# B&R Automation Studio project 3964r
Automation Studio 4.2.8.54 SP

## Configuration cp1381

CPU X20CP1381, AutomationRuntime B4.26, Build 4.1.2, Vc V4.26.2

CPU X20CP3586, AutomationRuntime B4.26, Build 4.1.2, Vc V4.26.2

### Task classes (Cpu.sw)
```
Cyclic#1 (cycle 10000 us, tolerance 10000 us):
  3964r1 <- 3964r.prg
Binaries: TCData, arconfig, asfw, ashwd, iomap, asnxdb1, User, Role, sysconf
Libraries: DRV_3964, dvframe, runtime, asstring, standard, astime, asieccon, IecCheck, sys_lib, AsBrStr
```

### Hardware
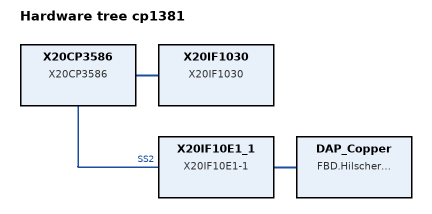
```
DAP_Copper : FBD.Hilscher.PNIOGenDevDTM2.DAP Copper.V1.09.05 v1.9.5 (OrderNumber=DAP Copper)  [PN1 -> X20IF10E1_1.IF1 (NodeNumber=1)]
  DtmId = 207df88f-8d0b-476b-a90a-ff4e51565477
  DtmRef = FBD.Hilscher.PNIOGenDevDTM2.DAP Copper.V1.09.05
  ChannelBlocks_54764a2b-737d-4760-b2ae-f15fab32f69c  // Retrofit Image <Slot 1>
  IO_InputImage_54764a2b-737d-4760-b2ae-f15fab32f69c
  IO_OutputImage_54764a2b-737d-4760-b2ae-f15fab32f69c
X20CP3586 : X20CP3586 v1.3.2.0
  Connector IF2:
    ActivateDevice = 1
    EthInterfaceRedundant = 0
    Mode = Manual
    InternetAddress = 192.168.20.10
    SubnetMask = 255.255.255.0
  Connector IF3:
    EplInterfaceRedundant = 0
    CycleTime = 10000
    EplEthInterfaceRedundant = 0
  ConfigurationID = test1_cp1381
  TimerDeviceType = SWIOTIMER
  Cyclic1Duration = 10000
  Cyclic1Tolerance = 10000
  Cyclic2Duration = 20000
  Cyclic2Tolerance = 20000
  Cyclic3Duration = 10000
  Cyclic3Tolerance = 50000
  Cyclic4Duration = 100000
  Cyclic4Tolerance = 100000
  Cyclic5Duration = 200000
  Cyclic5Tolerance = 200000
  Cyclic6Duration = 500000
  Cyclic6Tolerance = 500000
  Cyclic7Duration = 1000000
  Cyclic7Tolerance = 1000000
  Cyclic8Duration = 10000
  Cyclic8Tolerance = 30000000
X20IF1030 : X20IF1030 v1.1.7.0  [SS -> X20CP3586.SS1]
X20IF10E1_1 : X20IF10E1-1 v1.1.5.0  [SS -> X20CP3586.SS2]
  Connector IF1:
    DtmRef = FBDIF.Hilscher.PNIOControllerDTM2.NETX 100 RE/PNM
    DtmId = 1afa87f6-e739-4a4c-a598-27084086dda1
  ConfigFile = X20IF10E1_1.dtm
  ConfigModule = asnxdb1
```

### IoMap.iom - X20CP3586/IoMap.iom
```iecst
VAR_CONFIG
	::3964r1:profinetInput1[0] AT %IB."DAP_Copper".Module001_Input8_00;
	::3964r1:profinetInput1[1] AT %IB."DAP_Copper".Module001_Input8_01;
	::3964r1:profinetInput1[2] AT %IB."DAP_Copper".Module001_Input8_02;
	::3964r1:profinetInput1[3] AT %IB."DAP_Copper".Module001_Input8_03;
	::3964r1:profinetOutput1[0] AT %QB."DAP_Copper".Module001_Output8_00;
	::3964r1:profinetOutput1[1] AT %QB."DAP_Copper".Module001_Output8_01;
	::3964r1:profinetOutput1[2] AT %QB."DAP_Copper".Module001_Output8_02;
	::3964r1:profinetOutput1[3] AT %QB."DAP_Copper".Module001_Output8_03;
	::3964r1:profinetInput2[0] AT %IB."DAP_Copper".Module001_Input_00;
	::3964r1:profinetInput2[1] AT %IB."DAP_Copper".Module001_Input_01;
	::3964r1:profinetInput2[2] AT %IB."DAP_Copper".Module001_Input_02;
	::3964r1:profinetInput2[3] AT %IB."DAP_Copper".Module001_Input_03;
	::3964r1:profinetInput2[4] AT %IB."DAP_Copper".Module001_Input_04;
	::3964r1:profinetInput2[5] AT %IB."DAP_Copper".Module001_Input_05;
	::3964r1:profinetInput2[6] AT %IB."DAP_Copper".Module001_Input_06;
	::3964r1:profinetInput2[7] AT %IB."DAP_Copper".Module001_Input_07;
	::3964r1:profinetInput2[8] AT %IB."DAP_Copper".Module001_Input_08;
	::3964r1:profinetInput2[9] AT %IB."DAP_Copper".Module001_Input_09;
	::3964r1:profinetInput2[10] AT %IB."DAP_Copper".Module001_Input_10;
	::3964r1:profinetOutput2[0] AT %QB."DAP_Copper".Module001_Output_00;
	::3964r1:profinetOutput2[1] AT %QB."DAP_Copper".Module001_Output_01;
	::3964r1:profinetOutput2[2] AT %QB."DAP_Copper".Module001_Output_02;
	::3964r1:profinetOutput2[3] AT %QB."DAP_Copper".Module001_Output_03;
	::3964r1:profinetOutput2[4] AT %QB."DAP_Copper".Module001_Output_04;
	::3964r1:profinetOutput2[5] AT %QB."DAP_Copper".Module001_Output_05;
	::3964r1:profinetOutput2[6] AT %QB."DAP_Copper".Module001_Output_06;
	::3964r1:profinetOutput2[7] AT %QB."DAP_Copper".Module001_Output_07;
	::3964r1:profinetOutput2[8] AT %QB."DAP_Copper".Module001_Output_08;
	::3964r1:profinetOutput2[9] AT %QB."DAP_Copper".Module001_Output_09;
	::3964r1:profinetOutput2[10] AT %QB."DAP_Copper".Module001_Output_10;
END_VAR
```

## Logical view

Binary libraries used (declarations not repeated): operator, runtime, astime, AsIecCon, DRV_3964, dvframe, asstring, standard, sys_lib, AsBrStr

### Package Logical/Libraries - Global libraries

### Library Logical/Libraries/IecCheck (IEC)
Depends on: sys_lib, AsBrStr

### Program Logical/3964r (IEC)

#### Types.typ
```iecst
TYPE
	FromFronius : 	STRUCT
		arcStable : BOOL;
		processActive : BOOL;
		mainCurrentSignal : BOOL;
		torchCollisionProtection : BOOL;
		powerSourceReady : BOOL;
		communicationReady : BOOL;
		powerOutsideRange : BOOL;
		weldingVoltageActual : UINT;
		weldingCurrentActual : UINT;
		wireFeedSpeed : UINT;
	END_STRUCT;
	FromComau : 	STRUCT
		weldingStart : BOOL;
		robotReady : BOOL;
		modesBit0 : BOOL;
		modesBit1 : BOOL;
		modesBit2 : BOOL;
		gasTest : BOOL;
		wireInching : BOOL;
		wireRetract : BOOL;
		touchSensing : BOOL;
		torchBlowOut : BOOL;
		jobNumber : USINT;
		weldingSimulation : BOOL;
		powerCommand : UINT;
		arcLengthCorrection : UINT;
		pulseCorrection : USINT;
		burnBackCommand : USINT;
		synchroPulseDisable : BOOL;
		temp : ARRAY[0..19]OF USINT;
	END_STRUCT;
	Interface3964R : 	STRUCT
		fromComau : FromComau;
		fromFronius : FromFronius;
	END_STRUCT;
END_TYPE
```

#### Variables.var
```iecst
VAR
	interface3964R : Interface3964R;
	step : INT;
	FRM_xopen_0 : FRM_xopen;
	FRM_read_0 : FRM_read;
	dataRead : ARRAY[0..19] OF USINT;
	FRM_rbuf_0 : FRM_rbuf;
	dataReadLength : INT;
	FRM_gbuf_0 : FRM_gbuf;
	FRM_write_0 : FRM_write;
	dataWrite : ARRAY[0..19] OF USINT;
	dataWriteLenght : INT;
	xopenconfig : XOPENCONFIG;
	BCC : USINT;
	i : INT;
	telegramType : USINT;
	stepOld : INT;
	profinetInput1 : ARRAY[0..3] OF USINT;
	profinetInput2 : ARRAY[0..10] OF USINT;
	profinetOutput1 : ARRAY[0..3] OF USINT;
	profinetOutput2 : ARRAY[0..10] OF USINT;
END_VAR
```

#### Cyclic.st
```iecst
PROGRAM _CYCLIC

	(* read data from new Fronius *)
	interface3964R.fromFronius.arcStable := profinetInput1[0].0;
	interface3964R.fromFronius.processActive := profinetInput1[0].2;
	interface3964R.fromFronius.mainCurrentSignal := profinetInput1[0].3;
	interface3964R.fromFronius.torchCollisionProtection := profinetInput1[0].4;
	interface3964R.fromFronius.powerSourceReady := profinetInput1[0].5;
	interface3964R.fromFronius.communicationReady := profinetInput1[0].6;
	interface3964R.fromFronius.powerOutsideRange := profinetInput1[3].7;

	interface3964R.fromFronius.weldingVoltageActual := profinetInput2[0] + 256*profinetInput2[1];
	interface3964R.fromFronius.weldingCurrentActual := profinetInput2[2] + 256*profinetInput2[3];
	interface3964R.fromFronius.wireFeedSpeed := profinetInput2[8] + 256*profinetInput2[9];

	(* communication with robot via protocol 3964r *)
	REPEAT
		stepOld := step;

		CASE step OF
			0:
				xopenconfig.rx_cnt := 1;
				xopenconfig.tx_cnt := 1;

				FRM_xopen_0.enable := TRUE;
				FRM_xopen_0.device := ADR('SS1.IF1');
				//			FRM_xopen_0.device := ADR('IF6.ST1.IF1');
				FRM_xopen_0.mode := ADR('/PHY=RS422 /BD=38400 /PA=E /DB=8 /SB=1');
				FRM_xopen_0.config := ADR(xopenconfig);

				FRM_xopen_0();

				IF FRM_xopen_0.status = 0 THEN
					step := 1;
				END_IF

			1:
				FRM_read_0.enable := TRUE;
				FRM_read_0.ident := FRM_xopen_0.ident;
				FRM_read_0();

				IF FRM_read_0.status = 0 THEN
					step := step + 1;
				END_IF

			2:
				dataReadLength := MIN(FRM_read_0.buflng, SIZEOF(dataRead));
				memcpy(ADR(dataRead), FRM_read_0.buffer, dataReadLength);

				FRM_rbuf_0.enable := TRUE;
				FRM_rbuf_0.ident := FRM_xopen_0.ident;
				FRM_rbuf_0.buffer := FRM_read_0.buffer;
				FRM_rbuf_0.buflng := dataReadLength;
				FRM_rbuf_0();

				IF FRM_rbuf_0.status = 0 THEN
					step := step + 1;
				END_IF

			3:
				IF dataReadLength = 1 AND dataRead[0] = 16#02 THEN
					step := step + 1;
				ELSE
					step := 1;
				END_IF

			4:
				FRM_gbuf_0.enable := TRUE;
				FRM_gbuf_0.ident := FRM_xopen_0.ident;
				FRM_gbuf_0();

				IF FRM_gbuf_0.status = 0 THEN
					step := step + 1;
				END_IF

			5:
				dataWrite[0] := 16#10;
				dataWriteLenght := 1;

				memcpy(FRM_gbuf_0.buffer, ADR(dataWrite), dataWriteLenght);

				FRM_write_0.enable := TRUE;
				FRM_write_0.ident := FRM_xopen_0.ident;
				FRM_write_0.buffer := FRM_gbuf_0.buffer;
				FRM_write_0.buflng := dataWriteLenght;
				FRM_write_0();

				IF FRM_write_0.status = 0 THEN
					step := step + 1;
				END_IF

			6:
				FRM_read_0.enable := TRUE;
				FRM_read_0.ident := FRM_xopen_0.ident;
				FRM_read_0();

				IF FRM_read_0.status = 0 THEN
					step := step + 1;
				END_IF

			7:
				dataReadLength := MIN(FRM_read_0.buflng, SIZEOF(dataRead));
				memcpy(ADR(dataRead), FRM_read_0.buffer, dataReadLength);

				FRM_rbuf_0.enable := TRUE;
				FRM_rbuf_0.ident := FRM_xopen_0.ident;
				FRM_rbuf_0.buffer := FRM_read_0.buffer;
				FRM_rbuf_0.buflng := dataReadLength;
				FRM_rbuf_0();

				IF FRM_rbuf_0.status = 0 THEN
					step := step + 1;
				END_IF

			8:
				IF dataReadLength > 1 THEN
					//compute checksum
					BCC := 0;
					FOR i:= 0 TO dataReadLength - 2 DO
						BCC := BCC XOR dataRead[i];
					END_FOR
					IF BCC = dataRead[dataReadLength - 1] THEN
						CASE dataRead[0] OF
							1:
								interface3964R.fromComau.temp := dataRead;

								interface3964R.fromComau.weldingStart := dataRead[1].0;
								interface3964R.fromComau.robotReady := dataRead[1].1;
								interface3964R.fromComau.modesBit0 := dataRead[1].2;
								interface3964R.fromComau.modesBit1 := dataRead[1].3;
								interface3964R.fromComau.modesBit2 := dataRead[1].4;
								interface3964R.fromComau.gasTest := dataRead[2].0;
								interface3964R.fromComau.wireInching := dataRead[2].1;
								interface3964R.fromComau.wireRetract := dataRead[2].2;
								interface3964R.fromComau.touchSensing := dataRead[2].4;
								interface3964R.fromComau.torchBlowOut := dataRead[2].5;
								interface3964R.fromComau.jobNumber := dataRead[3];
								interface3964R.fromComau.weldingSimulation := dataRead[4].7;
								interface3964R.fromComau.powerCommand := dataRead[5] + 256*dataRead[6];
								interface3964R.fromComau.arcLengthCorrection := dataRead[7] + 256*dataRead[8];
								interface3964R.fromComau.pulseCorrection := dataRead[9];
								interface3964R.fromComau.burnBackCommand := dataRead[10];
								interface3964R.fromComau.synchroPulseDisable := dataRead[11].0;

							ELSE

						END_CASE
						telegramType := dataRead[0];
						step := step + 1;
					ELSE
						step := 1;
					END_IF
				ELSE
					step := 1;
				END_IF

			9:
				FRM_gbuf_0.enable := TRUE;
				FRM_gbuf_0.ident := FRM_xopen_0.ident;
				FRM_gbuf_0();

				IF FRM_gbuf_0.status = 0 THEN
					step := step + 1;
				END_IF

			10:
				dataWrite[0] := 16#10;
				dataWrite[1] := 16#2;
				dataWriteLenght := 2;

				CASE telegramType OF
					4:
						dataWrite[2] := 16#04;
						dataWrite[3].0 := interface3964R.fromFronius.arcStable;//16#40;
						dataWrite[3].2 := interface3964R.fromFronius.processActive;
						dataWrite[3].3 := interface3964R.fromFronius.mainCurrentSignal;
						dataWrite[3].4 := interface3964R.fromFronius.torchCollisionProtection;
						dataWrite[3].5 := interface3964R.fromFronius.powerSourceReady;
						dataWrite[3].6 := interface3964R.fromFronius.communicationReady;
						dataWrite[4] := 0;
						dataWrite[5] := 0;
						dataWrite[6] := 0;
						dataWriteLenght := 7;
					5:
						dataWrite[2] := 16#05;
						dataWrite[3] := UINT_TO_USINT(interface3964R.fromFronius.weldingVoltageActual AND 16#FF);//16#55;
						dataWrite[4] := UINT_TO_USINT(SHR(interface3964R.fromFronius.weldingVoltageActual,8));//16#2E;
						dataWrite[5] := 0;//UINT_TO_USINT(interface3964R.fromFronius.weldingCurrentActual AND 16#FF);//16#B4;
						dataWrite[6] := 0;//UINT_TO_USINT(SHR(interface3964R.fromFronius.weldingCurrentActual,8));//16#08;

						dataWrite[7] := 0;
						dataWrite[8] := UINT_TO_USINT(interface3964R.fromFronius.wireFeedSpeed AND 16#FF);//16#C8;
						dataWrite[9] := UINT_TO_USINT(SHR(interface3964R.fromFronius.wireFeedSpeed,8));//0;
						dataWriteLenght := 10;
					ELSE
						dataWrite[2] := 16#06;
						dataWrite[3] := 16#00;
						dataWriteLenght := 4;
				END_CASE

				//add 16#10, 16#03
				dataWrite[dataWriteLenght] := 16#10;
				dataWrite[dataWriteLenght+1] := 16#03;

				//add checksum
				BCC := 0;
				FOR i:= 2 TO dataWriteLenght + 1 DO
					BCC := BCC XOR dataWrite[i];
				END_FOR
				dataWrite[dataWriteLenght+2] := BCC;
				dataWriteLenght := dataWriteLenght + 3;

				memcpy(FRM_gbuf_0.buffer, ADR(dataWrite), dataWriteLenght);

				FRM_write_0.enable := TRUE;
				FRM_write_0.ident := FRM_xopen_0.ident;
				FRM_write_0.buffer := FRM_gbuf_0.buffer;
				FRM_write_0.buflng := dataWriteLenght;
				FRM_write_0();

				IF FRM_write_0.status = 0 THEN
					step := 1;
				END_IF

		END_CASE

		UNTIL step = stepOld

	END_REPEAT

	(* write data to Fronius *)
	profinetOutput1[0].0 := interface3964R.fromComau.weldingStart;
	profinetOutput1[0].1 := interface3964R.fromComau.robotReady;
	profinetOutput1[0].2 := interface3964R.fromComau.modesBit0;
	profinetOutput1[0].3 := interface3964R.fromComau.modesBit1;
	profinetOutput1[0].4 := interface3964R.fromComau.modesBit2;
	profinetOutput1[1].0 := interface3964R.fromComau.gasTest;
	profinetOutput1[1].1 := interface3964R.fromComau.wireInching;
	profinetOutput1[1].2 := interface3964R.fromComau.wireRetract;
	profinetOutput1[1].4 := interface3964R.fromComau.touchSensing;
	profinetOutput1[1].5 := interface3964R.fromComau.torchBlowOut;
	profinetOutput1[2] := interface3964R.fromComau.jobNumber;
	profinetOutput1[3].7 := interface3964R.fromComau.weldingSimulation;

	profinetOutput2[0] := UINT_TO_USINT(interface3964R.fromComau.powerCommand AND 16#FF);
	profinetOutput2[1] := UINT_TO_USINT(SHR(interface3964R.fromComau.powerCommand, 8));
	profinetOutput2[2] := UINT_TO_USINT(interface3964R.fromComau.arcLengthCorrection AND 16#FF);
	profinetOutput2[3] := UINT_TO_USINT(SHR(interface3964R.fromComau.arcLengthCorrection, 8));
	profinetOutput2[4] := interface3964R.fromComau.pulseCorrection;
	profinetOutput2[6] := interface3964R.fromComau.burnBackCommand;
	profinetOutput2[10].0 := interface3964R.fromComau.synchroPulseDisable;

END_PROGRAM
```

### Program Logical/Program (IEC)

#### Main.st - Cyclic code
```iecst
PROGRAM _INIT
	(* Insert code here *)

END_PROGRAM

PROGRAM _CYCLIC
	CASE step OF
		0:
			S39SOpen_0.enable := TRUE;
			S39SOpen_0.pDevice := ADR('IF6.ST1.IF1');
			S39SOpen_0.pMode := ADR('/PHY=RS422 /BD=38400 /PA=E /DB=8 /SB=1');
			S39SOpen_0.rk512 := FALSE;
			S39SOpen_0.buflen := 280;
			S39SOpen_0.timeout := 0;
			S39SOpen_0.retry := 0;

			S39SOpen_0();

			IF S39SOpen_0.status = 0 THEN
				step := 1;
			END_IF

		1:
			rxBuffer ACCESS S39SOpen_0.rx_buf;
			txBuffer ACCESS S39SOpen_0.tx_buf;

			S39Slave_0.enable := TRUE;
			S39Slave_0.ident := S39SOpen_0.ident;
			S39Slave_0.mode := s39MODE_SEND_RECV;//s39MODE_RECV_ONLY;//s39MODE_SEND_RECV;
			S39Slave_0();

	END_CASE

END_PROGRAM
```

### Program Logical/Program1

#### Variables.var
```iecst
VAR
	step : INT;
	S39SOpen_0 : S39SOpen;
	S39Slave_0 : S39Slave;
	txBuffer : REFERENCE TO ARRAY[0..279] OF BYTE;
	rxBuffer : REFERENCE TO ARRAY[0..279] OF BYTE;
END_VAR
```

#### Main.st
```iecst
PROGRAM _INIT
	(* Insert code here *)

END_PROGRAM

PROGRAM _CYCLIC
	CASE step OF
		0:
			S39SOpen_0.enable := TRUE;
			S39SOpen_0.pDevice := ADR('IF6.ST1.IF1');
			S39SOpen_0.pMode := ADR('/PHY=RS422 /BD=38400 /PA=E /DB=8 /SB=1');
			S39SOpen_0.rk512 := FALSE;
			S39SOpen_0.buflen := 280;
			S39SOpen_0.timeout := 0;
			S39SOpen_0.retry := 0;

			S39SOpen_0();

			IF S39SOpen_0.status = 0 THEN
				step := 1;
			END_IF

		1:
			rxBuffer ACCESS S39SOpen_0.rx_buf;
			txBuffer ACCESS S39SOpen_0.tx_buf;

			S39Slave_0.enable := TRUE;
			S39Slave_0.ident := S39SOpen_0.ident;
			S39Slave_0.mode := s39MODE_SEND_ONLY;//s39MODE_RECV_ONLY;//s39MODE_SEND_RECV;
			S39Slave_0();

	END_CASE

END_PROGRAM
```

Listed in the project but not available here: Logical/Global.typ, Logical/Global.var, Logical/Libraries/IecCheck/IecCheck.fun, Logical/Libraries/IecCheck/IecCheck.st, Logical/Program/Types.typ, Logical/Program/Variables.var
